{attribute addProperty BoxType "AX8206-0000-0041-0041"}
{attribute addProperty Id "Ch_B_AxisMain_InputsCh_B_AxisMain_Inputs_F44016C911214Ch_B_AxisMain_OutputsCh_B_AxisMain_Outputs_3FCFC8F5162Ch_B_Interpolator_OutputsCh_B_Interpolator_Outputs_EA1B41E0648Ch_B_PositionControl_InputsCh_B_PositionControl_Inputs_61BD0E57324Ch_B_TorqueControl_OutputsCh_B_TorqueControl_Outputs_0381A30F162"}
{attribute addProperty CRC "1572996527"}
{attribute addProperty SizeInBites "240"}
{attribute addProperty SizeInBytes "30"}
TYPE Ch_B_5DC205AF :
STRUCT
	{attribute addProperty Name "Ch_B_AxisMain_Inputs"}
	Ch_B_AxisMain_Inputs  : Ch_B_AxisMain_Inputs_F44016C9;
	{attribute addProperty Name "Ch_B_AxisMain_Outputs"}
	Ch_B_AxisMain_Outputs  : Ch_B_AxisMain_Outputs_3FCFC8F5;
	{attribute addProperty Name "Ch_B_Interpolator_Outputs"}
	Ch_B_Interpolator_Outputs  : Ch_B_Interpolator_Outputs_EA1B41E0;
	{attribute addProperty Name "Ch_B_PositionControl_Inputs"}
	Ch_B_PositionControl_Inputs  : Ch_B_PositionControl_Inputs_61BD0E57;
	{attribute addProperty Name "Ch_B_TorqueControl_Outputs"}
	Ch_B_TorqueControl_Outputs  : Ch_B_TorqueControl_Outputs_0381A30F;
END_STRUCT
END_TYPE

(* stored: Version 1.2.0.0, ProductVersion 3.1.4024.9
   DUT Ch_B_5DC205AF: Id {7dac8771-b98d-4464-acc9-bce9b23c3e7c} *)
